FUNCTION_BLOCK horimetro (* Composite Function Block Type *)
  (* Standard: 61499-2 *)
  (* Version 0.0, 14/01/2026, Schneider Electric, template *)
  PACKAGE Hidryco.HidrycoLib;
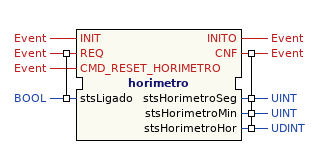
  EVENT_INPUT
    INIT; (* Initialization Request *)
    REQ WITH stsLigado; (* Normal Execution Request *)
    CMD_RESET_HORIMETRO;
  END_EVENT
  EVENT_OUTPUT
    INITO; (* Initialization Confirm *)
    CNF WITH stsHorimetroSeg, stsHorimetroMin, stsHorimetroHor; (* Execution Confirmation *)
  END_EVENT
  VAR_INPUT
    stsLigado : BOOL;
  END_VAR
  VAR_OUTPUT
    stsHorimetroSeg : UINT;
    stsHorimetroMin : UINT;
    stsHorimetroHor : UDINT;
  END_VAR
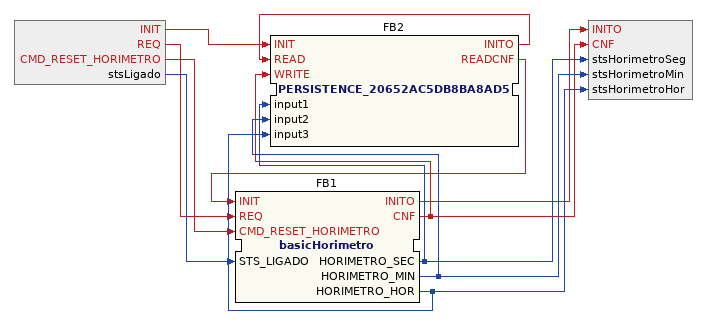
  FBS
    FB1 : basicHorimetro;
    FB2 : PERSISTENCE_20652AC5DB8BA8AD5; {SET_ATTRIBUTE(Configuration.GenericFBType.InterfaceParams, Runtime.Standard#I:=3;input${I$}:UINT,UINT,UDINT)}
  END_FBS
  EVENT_CONNECTIONS
    REQ TO FB1.REQ;
    FB1.CNF TO CNF;
    CMD_RESET_HORIMETRO TO FB1.CMD_RESET_HORIMETRO;
    FB1.INITO TO INITO;
    INIT TO FB2.INIT;
    FB2.INITO TO FB2.READ;
    FB1.CNF TO FB2.WRITE;
    FB2.READCNF TO FB1.INIT;
  END_CONNECTIONS
  DATA_CONNECTIONS
    stsLigado TO FB1.STS_LIGADO;
    FB1.HORIMETRO_HOR TO stsHorimetroHor;
    FB1.HORIMETRO_MIN TO stsHorimetroMin;
    FB1.HORIMETRO_SEC TO stsHorimetroSeg;
    FB1.HORIMETRO_SEC TO FB2.input1;
    FB1.HORIMETRO_MIN TO FB2.input2;
    FB1.HORIMETRO_HOR TO FB2.input3;
  END_CONNECTIONS
END_FUNCTION_BLOCK
